PROGRAM P_RunClock

VAR
	fbRunClock : FB_RunClock; 
END_VAR

// Runs FB with given values
fbRunClock(
	bStart := TRUE,
	bStop := G_Inputs.bStopButton, // Stop button on controller
	fCycleTime := G_Parameter.fCycleTime, // Time step
	
	fTime => G_OPC.fTime // Output time 
);

END_PROGRAM

(* stored: Version 1.1.0.1
   POU P_RunClock: Id {d8c930b5-bf90-4658-99e0-6b7148646632}, SpecialFunc None *)
